// TIA Portal V18 export
DATA_BLOCK "Var"   // DB1
{ S7_Optimized_Access := 'FALSE' }
VERSION : 0.1
// stored: AutoNumber true, IsOnlyStoredInLoadMemory false, IsWriteProtectedInAS false
   VAR RETAIN
      high_level_switch : Bool;
      panel_emergency_stop : Bool;
      pendant_emergency_stop : Bool;
      start_button : Bool;
      stop_button : Bool;
      FCV_valve_closed : Bool;
      FCV_valve_open : Bool;
      ESD_valve_closed : Bool;
      ESD_Valve_open : Bool;
      ground_signal1 : Bool;
      ground_signal2 : Bool;
      ESD_solenoid_valve_command : Bool;
      flowmeter_signal_Input : Int;
      flow_control_valve_output : Int;
      RTD_PT100_INPUT_1 : Int;
      RTD_PT100_INPUT_2 : Int;
      RTD_PT100_INPUT_3 : Int;
      Temperature : Int := 0;
      Temperature_threshold : Int := 100;
      Interlocks_idle : Bool;
      Grounding : Bool;
      In_loading : Bool;
      In_Draining : Bool;
      loaded_quantity : Real;
      Ready_to_Load : Bool;
      working_seq : Int;
      flow_meter_reset : Bool;
      "HSC_DATA.EdgeCount_real" : Real;
      "counter" : DInt;
      counter_real : Real;
      reset_counter : Bool;
      set_quantity : Int := 100;
      emergency_state : Bool;
      draining_flag : Bool;
      pump_signal : Bool;
      interlocks_loading : Bool;
      emergency_flag : Bool := false;
      instat_flowrate : Int;
      pause_flag : Bool;
      loading_flag : Bool;
      idle_flag : Bool;
      temperature_is_ok : Bool;
      drain_time_integer : Int := 10000;
      drain_time_time : Time := T#10000ms;
      drain_time_integer_seconds : Int := 10;
      Elapsed_drain_time : Int;
      Number_of_IBC : Int;
      Total_quantity : Real;
      lotto_terminato : Bool;
      freeze_counter : Bool;
      no_flow_states : Bool;
      FCV_low_flow_signal : Int := 5;
      FCV_high_flow_signal : Int := 10;
      quantity_of_LH_flow_intitial : Int := 20;
      quantity_of_LH_flow_percentage_initial : Int;
      quantity_of_HL_flow_final : Int := 20;
      quantity_of_HL_flow_percentage_final : Int;
      time_remained : Int;
      remained_quantity : Int;
      pulse_temp : DInt;
      recent_loaded_quantity : Int;
      No_of_IBC_all_time : Int;
   END_VAR
BEGIN
END_DATA_BLOCK
